KUKA KRL program: mixsort_place_select.src, mixsort_place_select.dat

--- mixsort_place_select.src ---
&ACCESS RVO1
&REL 22
&COMMENT Place Select
&PARAM DISKPATH = KRC:\R1\Program\MixSortMain
def mixsort_place_select()
;***********************************************************
;
; Copyright 2018 - 2024 speedbot All Rights reserved.
;
; File Name: mixsort_place_select.src
;
; Description:
;   Language             ==   Krl for KUKA ROBOT
;   Date                 ==   2022 - 06 - 27
;   Modification Data    ==   2024 - 10 - 25
;
; Author: speedbot
;
; Version: 1.1
;***********************************************************
    CopyPartData = AgentData.PartData

    if not MixPkCfg.BoxOrConv then
        switch CopyPartData.PlaceId
        case 1
            mixsort_drop01()
        case 2
            mixsort_drop02()
        case 3
            mixsort_drop03()
        case 3
            mixsort_drop04()
        default
            Offset = 0
            swrite(Msg[], State, Offset, "PlaceId Error[PlaceId:%D, MaxPlaceId:%D]", CopyPartData.PlaceId, MixPkCfg.NumPlPoint)
            err_write_("Mixsort", Msg[], true)
        endswitch
    else
        switch CopyPartData.PlaceId
        case 1
            mixsort_place01()
        case 2
            mixsort_place02()
        case 3
            mixsort_place03()
        case 4
            mixsort_place04()
        case 5
            mixsort_place05()
        case 6
            mixsort_place06()
        case 7
            mixsort_place07()
        case 8
            mixsort_place08()
        default
            Offset = 0
            swrite(Msg[], State, Offset, "PlaceId Error[PlaceId:%D, MaxPlaceId:%D]", CopyPartData.PlaceId, MixPkCfg.NumPlPoint)
            err_write_("Mixsort", Msg[], true)
        endswitch
    endif

end

--- mixsort_place_select.dat ---
&ACCESS RVO1
&REL 22
&COMMENT Place Select
&PARAM DISKPATH = KRC:\R1\Program\MixSortMain
defdat mixsort_place_select
;***********************************************************
;
; Copyright 2018 - 2024 speedbot All Rights reserved.
;
; File Name: mixsort_place_select.dat
;
; Description:
;   Language             ==   Krl for KUKA ROBOT
;   Date                 ==   2022 - 06 - 28
;   Modification Data    ==   2022 - 06 - 28
;
; Author: speedbot
;
; Version: 1.0
;***********************************************************


EXT  mixsort_place01()
EXT  mixsort_place02()
EXT  mixsort_place03()
EXT  mixsort_place04()
EXT  mixsort_place05()
EXT  mixsort_place06()
EXT  mixsort_place07()
EXT  mixsort_place08()
EXT  mixsort_drop01()
EXT  mixsort_drop02()
EXT  mixsort_drop03()
EXT  mixsort_drop04()

decl state_t State
decl int Offset = 0
decl char Msg[256]

DECL part_data_t CopyPartData

enddat
